FUNCTION_BLOCK FB_TibberAPI
//Tested and works with 4024.22 4024.29 4024.32 4024.35
//Will not work with any 4022. 4024.7 may also not work.
//Based on the Beckhoff Postman POST example: https://infosys.beckhoff.com/content/1033/tf6760_tc3_iot_https_rest/7876792971.html?id=8531523618449441037
VAR_INPUT
    bSend				: BOOL;
	pTibberPrice		: PVOID;
	nSize				: UINT;
	sToken				: STRING;
	eQuery				: E_Query;
END_VAR
VAR_IN_OUT
    fbClient            : FB_IotHttpClient;
END_VAR
VAR_OUTPUT
    bBusy               : BOOL;
    bError              : BOOL;
	nStatus				: UINT;
END_VAR
VAR
    fbRequest           : FB_IotHttpRequest;
	fbHeader            : FB_IotHttpHeaderFieldMap;
    fbJson              : FB_JsonDomParser;
	fbJsonDataType		: FB_JsonReadWriteDataType;
	RisingEdge          : R_TRIG; 
    sContent            : STRING (4095);
	sContentReceive		: STRING (6143);
    nErrCount           : UDINT;
	nState              : UDINT;
END_VAR

RisingEdge(CLK:= bSend);
CASE nState OF
0:
    IF RisingEdge.Q THEN
		sToken := CONCAT('Bearer	', sToken);
		fbHeader.AddField('Authorization', sToken, FALSE);
		fbRequest.sContentType := 'application/json; charset=utf-8';
		sContent := M_QueryType(eQuery := eQuery);
        IF fbRequest.SendRequest(sUri:= '/v1-beta/gql/', fbClient:= fbClient, eRequestType:= ETcIotHttpRequestType.HTTP_POST, pContent:= ADR(sContent), nContentSize:= LEN2(ADR(sContent)), fbHeader:=fbHeader) THEN
            nState:= 1;
            bBusy:= TRUE;
            bError:= FALSE;
        END_IF
    END_IF
1:	
	IF NOT fbRequest.bBusy THEN
		bError:= TRUE;
		IF NOT fbRequest.bError THEN				 					
			IF fbRequest.GetContent(pContent:= ADR(sContentReceive), nContentSize:= SIZEOF(sContentReceive), bSetNullTermination:= TRUE) AND fbRequest.nStatusCode >= 200 AND fbRequest.nStatusCode < 300 THEN
					IF fbJsonDataType.SetSymbolFromJson(sContentReceive, 'ST_TibberPrice', nSize, pTibberPrice) THEN
						bError:= FALSE;
					END_IF				
			END_IF				
		END_IF
		nState:= 0;
		nStatus := fbRequest.nStatusCode;
		bBusy:= FALSE;
		IF bError THEN
			nErrCount:= nErrCount+1;
		END_IF		
	END_IF  	
END_CASE

METHOD M_QueryType : STRING (4095)
VAR_INPUT
	eQuery		: E_Query;
END_VAR
CASE eQuery OF
	E_Query.current:
		M_QueryType:= '{ "query": "{viewer {homes {currentSubscription{priceInfo{current{total energy tax startsAt }}}}}}" }';
	E_Query.today:
		M_QueryType:= '{ "query": "{viewer {homes {currentSubscription {priceInfo {today {total energy tax startsAt }}}}}}" }';
	E_Query.tomorrow:
		M_QueryType:= '{ "query": "{viewer {homes {currentSubscription {priceInfo {tomorrow {total energy tax startsAt }}}}}}" }';
	E_Query.all:
		M_QueryType:= '{ "query": "{viewer {homes{currentSubscription {priceInfo {current {total energy tax startsAt}today {total energy tax startsAt}tomorrow {total energy tax startsAt }}}}}}" }';
END_CASE
END_METHOD

END_FUNCTION_BLOCK

(* stored: Version 1.1.0.1, ProductVersion 3.1.4024.11
   POU FB_TibberAPI: Id {a130465d-acc1-4978-9c98-c029987b13e7}, SpecialFunc None
   Method M_QueryType: Id {a5470e73-a6fe-4a9b-a87a-f5c9e170e702} *)
